// TIA Portal project "ControlMotor" (V15.1)
// En este trabajo se hace control de un motor dc para

(* hardware
DEVICE "S7-1200 station_1"  S7-1200 Station
   slot 0: "Rack_0"  S7-1200 Rack  Rack  V1.0
   slot 1: "PLC_1"  CPU 1214C AC/DC/Rly  6ES7 214-1BG40-0XB0  V4.2
   slot 3: "AQ 1x12BIT_1"  AQ1 signal board  6ES7 232-4HA30-0XB0  V1.0
*)

// ===== PLC "PLC_1"  CPU 1214C AC/DC/Rly =====

VAR_GLOBAL   // PLC tag table "Tabla de variables estándar"
   "Arranque" AT %I0.0 : Bool;
   "Parada" AT %I0.1 : Bool;
   "EN" AT %Q0.0 : Bool;
   "Norm_Taco" AT %MD1 : DWord;
   "Taco" AT %IW64 : Int;
   "Scale_Taco" AT %MD2 : Real;
   "Norm_Ref" AT %MD3 : Real;
   "Scale_Ref" AT %MD4 : Real;
   "Motor_Out" AT %QW80 : Int;
   "PID_Out" AT %MD10 : Real;
   "Ref" AT %IW66 : Int;
   "Tag_1" AT %MD100 : DWord;
END_VAR

ORGANIZATION_BLOCK "Main"   // OB1, LAD, ProgramCycle
TITLE = "Main Program Sweep (Cycle)"
{ S7_Optimized_Access := 'TRUE' }
VERSION : 0.1
   VAR_INPUT
      Initial_Call : Bool;   // Initial call of this OB
      Remanence : Bool;   // =True, if remanent data are available
   END_VAR
BEGIN

REGION Network 1: Pulsadores_Arranque_Parada
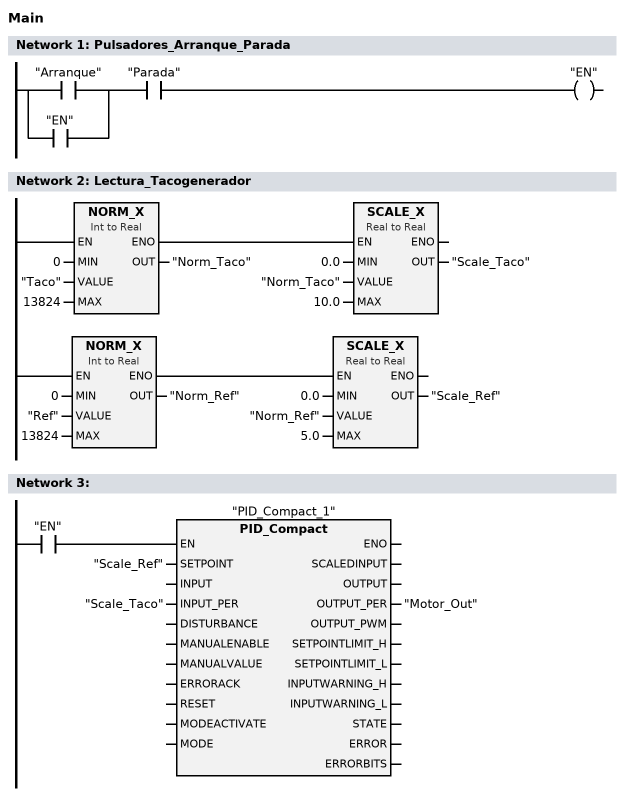
   RUNG wire#powerrail
      Contact( "Arranque" )
      wire#w1
      Contact( "Parada" )
      Coil( "EN" )
   END_RUNG
   RUNG wire#powerrail
      Contact( "EN" )
   END_RUNG wire#w1
   // the same network as SCL:
   "EN" := ("Arranque" OR "EN") AND "Parada";
END_REGION

REGION Network 2: Lectura_Tacogenerador
   RUNG wire#powerrail
      { S7_Templates := "[SrcType := Int, DestType := Real]" } Normalize(min := 0, value := "Taco", max := 13824, out => "Norm_Taco")
      { S7_Templates := "[SrcType := Real, DestType := Real]" } Scale(min := 0.0, value := "Norm_Taco", max := 10.0, out => "Scale_Taco")
   END_RUNG
   RUNG wire#powerrail
      { S7_Templates := "[SrcType := Int, DestType := Real]" } Normalize(min := 0, value := "Ref", max := 13824, out => "Norm_Ref")
      { S7_Templates := "[SrcType := Real, DestType := Real]" } Scale(min := 0.0, value := "Norm_Ref", max := 5.0, out => "Scale_Ref")
   END_RUNG
   // the same network as SCL:
   "Norm_Taco" := NORM_X(MIN := 0, VALUE := "Taco", MAX := 13824);
   "Scale_Taco" := SCALE_X(MIN := 0.0, VALUE := "Norm_Taco", MAX := 10.0);
   "Norm_Ref" := NORM_X(MIN := 0, VALUE := "Ref", MAX := 13824);
   "Scale_Ref" := SCALE_X(MIN := 0.0, VALUE := "Norm_Ref", MAX := 5.0);
END_REGION

REGION Network 3
   IF "EN" THEN
       "PID_Compact_1"(Setpoint := "Scale_Ref", Input_PER := "Scale_Taco", Output_PER => "Motor_Out");   // PID_Compact
   END_IF;
END_REGION
END_ORGANIZATION_BLOCK